Universal Robots PolyScope program: RQ_2FG_Pick&Place_Demo.urp

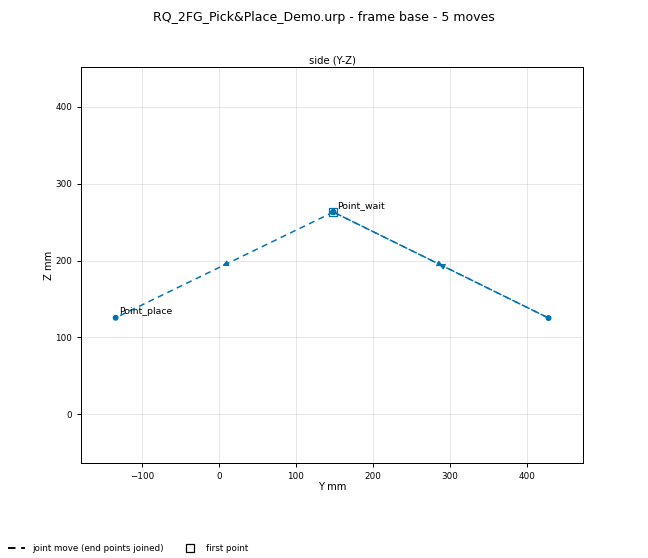
[picture p0: tool path of RQ_2FG_Pick&Place_Demo.urp in frame base, 5 of 5 moves have a stored position in this frame; points joined in program order, loops and branches not executed]
ProgramRoot directory=/home/ur/ursim-1.7_UR5/programs/Robotiq/2_Finger_Adaptive_Robot_Gripper/Examples; kinematics=(a=[0, -0.612, -0.5723, 0, 0, 0], d=[0.1273, 0, 0, 0.16394, 0.1157, 0.0922], alpha=[1.5708, 0, 0, 1.5708, -1.5708, 0], deltaTheta=[0, 0, 0, 0, 0, 0], status=notInitialized); name=RQ_2FG_Pick&Place_Demo; programVersion=(project__name=PolyScope, major__version=1, minor__version=7, svn__revision=9981, build__date=Feb 21 2013, 15:22:49); robotEnvironmentFileName=RQ_2FG_Installation
  MainProgram cartesianAcceleration=1.2; cartesianSpeed=0.25; jointAcceleration=1.3962634015954636; jointSpeed=1.0471975511965976; moveAsFastAsPossible=true; sharedProcessMoveBlendRadius=0.025; featureReference=(installationNameReference=Base); motionType=JOINT_SPACE
    Move cartesianAcceleration=1.2; cartesianSpeed=0.25; jointAcceleration=1.3962634015954636; jointSpeed=1.0471975511965976; moveAsFastAsPossible=true; sharedProcessMoveBlendRadius=0.025; featureReference=(installationNameReference=Base); motionType=JOINT_SPACE
      Waypoint blendRadius=0.05; cartesianAcceleration=1.2; cartesianSpeed=0.25; jointAcceleration=1.3962634015954636; jointSpeed=1.0471975511965976; nextMotionTime=2.0; stoppoint=true; useSharedBlendParameter=true; useSharedParameters=true; position=TCP in base x=422.585 y=148.572 z=263.039 mm, rx=-0.0012 ry=3.1163 rz=0.0389 rad; joints [33.397, -87.916, -118.071, -62.027, 90.404, 123.359] deg; positionType=FIXED_POSITION; waypointPoseInFeatureCoordinates=(pos=(x=0.42258461886856036, y=0.148572021533191, z=0.26303893099008774), rot=(x=-0.0012213597420371184, y=3.1162765268427233, z=0.038891918121804224)); name=Point_wait
    Script type=1; cachedFileContents=#Activation if not activated
      | if ((modbus_get_signal_status("Gripper_Status1", False) == False)  and (modbus_get_signal_status("Gripper_Status2", False) == False)):
      |     modbus_set_output_signal("Activate", True, False)
      | end
      | 
      | #Prohibit the movement
      | modbus_set_output_signal("Go_to_Requested", False, False)
      | while (modbus_get_signal_status("Action_Status", False) == True):
      |     sync()
      | end
      | 
      | #Awaiting the activation of the gripper
      | while (not(modbus_get_signal_status("Gripper_Status1", False) ==  True )):
      |     sync()
      | end
      | while (not(modbus_get_signal_status("Gripper_Status2", False) ==  True )):
      |     sync()
      | end; scriptFile=/home/ur/ursim-1.7_UR10/programs/Robotiq/2_Finger_Adaptive_Robot_Gripper/RQ_2FG_Activate_script.script
    While count=0; type=LOOP_FOREVER
      Move cartesianAcceleration=1.2; cartesianSpeed=0.25; jointAcceleration=1.3962634015954636; jointSpeed=1.0471975511965976; moveAsFastAsPossible=true; sharedProcessMoveBlendRadius=0.025; featureReference=(installationNameReference=Base); motionType=JOINT_SPACE
        Waypoint blendRadius=0.05; cartesianAcceleration=1.2; cartesianSpeed=0.25; jointAcceleration=1.3962634015954636; jointSpeed=1.0471975511965976; nextMotionTime=2.0; stoppoint=true; useSharedBlendParameter=true; useSharedParameters=true; position=TCP in base x=422.585 y=148.572 z=263.039 mm, rx=-0.0012 ry=3.1163 rz=0.0389 rad; joints [33.397, -87.916, -118.071, -62.027, 90.404, 123.359] deg; positionType=FIXED_POSITION; waypointPoseInFeatureCoordinates=(pos=(x=0.42258461886856036, y=0.148572021533191, z=0.26303893099008774), rot=(x=-0.0012213597420371184, y=3.1162765268427233, z=0.038891918121804224)); name=Point_wait
        Waypoint blendRadius=0.05; cartesianAcceleration=1.2; cartesianSpeed=0.25; jointAcceleration=1.3962634015954636; jointSpeed=1.0471975511965976; nextMotionTime=2.0; stoppoint=true; useSharedBlendParameter=true; useSharedParameters=true; position=TCP in base x=419.022 y=428.397 z=125.323 mm, rx=-0.0012 ry=3.1163 rz=0.0389 rad; joints [56.184, -117.85, -103.792, -46.37, 89.603, 146.132] deg; positionType=FIXED_POSITION; waypointPoseInFeatureCoordinates=(pos=(x=0.4190219316984625, y=0.42839680736151986, z=0.12532282398626846), rot=(x=-0.00122135974205825, y=3.1162765268427686, z=0.03889191812182904)); name=Point_pick
      CallSubProgram subProgramNodeToCall=255
      If expr=Contact_closing = True; type=IF_NODE
        Move cartesianAcceleration=1.2; cartesianSpeed=0.25; jointAcceleration=1.3962634015954636; jointSpeed=1.0471975511965976; moveAsFastAsPossible=true; sharedProcessMoveBlendRadius=0.025; featureReference=(installationNameReference=Base); motionType=JOINT_SPACE
          Waypoint blendRadius=0.05; cartesianAcceleration=1.2; cartesianSpeed=0.25; jointAcceleration=1.3962634015954636; jointSpeed=1.0471975511965976; nextMotionTime=2.0; stoppoint=true; useSharedBlendParameter=true; useSharedParameters=true; position=TCP in base x=422.585 y=148.572 z=263.039 mm, rx=-0.0012 ry=3.1163 rz=0.0389 rad; joints [33.397, -87.916, -118.071, -62.027, 90.404, 123.359] deg; positionType=FIXED_POSITION; waypointPoseInFeatureCoordinates=(pos=(x=0.42258461886856036, y=0.148572021533191, z=0.26303893099008774), rot=(x=-0.0012213597420371184, y=3.1162765268427233, z=0.038891918121804224)); name=Point_wait
          Waypoint blendRadius=0.05; cartesianAcceleration=1.2; cartesianSpeed=0.25; jointAcceleration=1.3962634015954636; jointSpeed=1.0471975511965976; nextMotionTime=2.0; stoppoint=true; useSharedBlendParameter=true; useSharedParameters=true; position=TCP in base x=428.356 y=-134.44 z=125.676 mm, rx=-0.0012 ry=3.1163 rz=0.0389 rad; joints [-3.641, -101.715, -128.085, -38.857, 91.519, 86.332] deg; positionType=FIXED_POSITION; waypointPoseInFeatureCoordinates=(pos=(x=0.42835576712717016, y=-0.1344399564428072, z=0.12567633989109042), rot=(x=-0.0012213598591346183, y=3.1162765318353176, z=0.03889191078463162)); name=Point_place
        CallSubProgram subProgramNodeToCall=0
      If type=ELSE_NODE
        CallSubProgram subProgramNodeToCall=0
  Thread name=Thread_1
    Script type=1; cachedFileContents=sync()
      | global RQ_2FG_Position=floor((modbus_get_signal_status("Position_Status",False))/256); scriptFile=/home/ur/ursim-1.7_UR10/programs/Robotiq/2_Finger_Adaptive_Robot_Gripper/RQ_2FG_Position_script.script
    Assignment assignmentValueSource=0; expr=RQ_2FG_Position; operatorValueType=INTEGER; valueSource=EXPRESSION; variable=(name=Grip_position, prefersPersistentValue=false, requestANewUniqueName=false)
  subProgramToCall file=/home/ur/ursim-1.7_UR10/programs/Robotiq/2_Finger_Adaptive_Robot_Gripper/RQ_2FG_Close.urp; name=SousP_RQ_2FG_Close
    Assignment assignmentValueSource=0; expr=255; operatorValueType=INTEGER; valueSource=EXPRESSION; variable=(name=Position_close, prefersPersistentValue=false, requestANewUniqueName=false)
    Assignment assignmentValueSource=0; expr=255; operatorValueType=INTEGER; valueSource=EXPRESSION; variable=(name=Speed_close, prefersPersistentValue=false, requestANewUniqueName=false)
    Assignment assignmentValueSource=0; expr=255; operatorValueType=INTEGER; valueSource=EXPRESSION; variable=(name=Force_close, prefersPersistentValue=false, requestANewUniqueName=false)
    Script type=1; cachedFileContents=#Allocation of modbus output registers with the desired settings
      | out_reg2_close = Speed_close * 256 + Force_close
      | modbus_set_output_register("Speed_Force_Req", out_reg2_close, False)
      | modbus_set_output_register("Position_Req", Position_close, False)
      | 
      | #Allow movement
      | modbus_set_output_signal("Go_to_Requested", True, False)
      | while(modbus_get_signal_status("Action_Status", False) == False):
      |     sync()
      | end
      | 
      | #Wait until the end of the movement
      | sleep(0.2)
      | while (not((modbus_get_signal_status("Obj_Det_Status1", False) == True) or (modbus_get_signal_status("Obj_Det_Status2", False) == True ))):
      |     sleep(0.1)
      |     sync()
      | end
      | 
      | sleep(0.2)
      | #Status check object detection
      | global obj_detect1 = modbus_get_signal_status("Obj_Det_Status1",False)
      | global obj_detect2 = modbus_get_signal_status("Obj_Det_Status2",False)
      | if ((obj_detect1 == False) and (obj_detect2 == True)):
      |     global Contact_opening = False
      |     global Contact_closing = True
      | else:
      |     if ((obj_detect1 == True) and (obj_detect2 == False)):
      |         global Contact_opening = True
      |         global Contact_closing = False
      |     else:
      |         global Contact_opening = False
      |         global Contact_closing = False
      |     end
      | end
      | 
      | #Prohibit the movement
      | modbus_set_output_signal("Go_to_Requested", False, False)
      | while(modbus_get_signal_status("Action_Status", False) == True):
      |     sync()
      | end; scriptFile=/home/ur/ursim-1.7_UR10/programs/Robotiq/2_Finger_Adaptive_Robot_Gripper/RQ_2FG_Close_script.script
  subProgramToCall file=/home/ur/ursim-1.7_UR10/programs/Robotiq/2_Finger_Adaptive_Robot_Gripper/RQ_2FG_Open.urp; name=SousP_RQ_2FG_Open
    Assignment assignmentValueSource=0; expr=0; operatorValueType=INTEGER; valueSource=EXPRESSION; variable=(name=Position_open, prefersPersistentValue=false, requestANewUniqueName=false)
    Assignment assignmentValueSource=0; expr=255; operatorValueType=INTEGER; valueSource=EXPRESSION; variable=(name=Speed_open, prefersPersistentValue=false, requestANewUniqueName=false)
    Assignment assignmentValueSource=0; expr=255; operatorValueType=INTEGER; valueSource=EXPRESSION; variable=(name=Force_open, prefersPersistentValue=false, requestANewUniqueName=false)
    Script type=1; cachedFileContents=#Allocation of modbus output registers with the desired settings
      | out_reg2_open = Speed_open * 256 + Force_open
      | modbus_set_output_register("Speed_Force_Req", out_reg2_open, False)
      | modbus_set_output_register("Position_Req", Position_open, False)
      | 
      | #Allow movement
      | modbus_set_output_signal("Go_to_Requested", True, False)
      | while(modbus_get_signal_status("Action_Status", False) == False):
      |     sync()
      | end
      | 
      | #Wait until the end of the movement
      | sleep(0.2)
      | while (not((modbus_get_signal_status("Obj_Det_Status1", False) == True) or (modbus_get_signal_status("Obj_Det_Status2", False) == True ))):
      |     sleep(0.1)
      |     sync()
      | end
      | 
      | sleep(0.2)
      | #Status check object detection
      | global obj_detect1 = modbus_get_signal_status("Obj_Det_Status1",False)
      | global obj_detect2 = modbus_get_signal_status("Obj_Det_Status2",False)
      | if ((obj_detect1 == False) and (obj_detect2 == True)):
      |     global Contact_opening = False
      |     global Contact_closing = True
      | else:
      |     if ((obj_detect1 == True) and (obj_detect2 == False)):
      |         global Contact_opening = True
      |         global Contact_closing = False
      |     else:
      |         global Contact_opening = False
      |         global Contact_closing = False
      |     end
      | end
      | 
      | #Prohibit the movement
      | modbus_set_output_signal("Go_to_Requested", False, False)
      | while(modbus_get_signal_status("Action_Status", False) == True):
      |     sync()
      | end; scriptFile=/home/ur/ursim-1.7_UR10/programs/Robotiq/2_Finger_Adaptive_Robot_Gripper/RQ_2FG_Open_script.script
